// TIA Portal V19 export
DATA_BLOCK "MANUAL"   // DB12
{ S7_Optimized_Access := 'TRUE' }
// stored: MemoryReserve 100
   VAR
      "MGF FEED PUMP WORKING" : Bool;
      "MFG FEED PUMP STANDBY" : Bool;
      "RO FEED PUMP WORKING" : Bool;
      "RO FEED PUMP STANDBY" : Bool;
      "RO HPP PUMP WORKING" : Bool;
      "RO HPP PUMP STANDBY" : Bool;
      "SMBS AGT-1" : Bool;
      "SALT TANK AGT-2" : Bool;
      "RO SMBS AGT-3" : Bool;
      "DP-1" : Bool;
      "DP-2" : Bool;
      "DP-3" : Bool;
      "DP-4" : Bool;
      "DP-5" : Bool;
      "DP-6" : Bool;
      "UV-1-DO" : Bool;
      "UV-2-DO" : Bool;
      HOOTER : Bool;
      "PSFV-1 – OPEN" : Bool;
      "PSFV-1 – CLOSE" : Bool;
      "PSFV-2 – OPEN" : Bool;
      "PSFV-2 – CLOSE" : Bool;
      "PSFV-3 – OPEN" : Bool;
      "PSFV-3 – CLOSE" : Bool;
      "PSFV-4 – OPEN" : Bool;
      "PSFV-4 – CLOSE" : Bool;
      "PSFV-5 – OPEN" : Bool;
      "PSFV-5 – CLOSE" : Bool;
      "PSFV-6 – OPEN" : Bool;
      "PSFV-6 – CLOSE" : Bool;
      "ACFV-1 – OPEN" : Bool;
      "ACFV-1 – CLOSE" : Bool;
      "ACFV-2 – OPEN" : Bool;
      "ACFV-2 – CLOSE" : Bool;
      "ACFV-3 – OPEN" : Bool;
      "ACFV-3 – CLOSE" : Bool;
      "ACFV-4 – OPEN" : Bool;
      "ACFV-4 - CLOSE" : Bool;
      "ACFV-5 – OPEN" : Bool;
      "ACFV-5 – CLOSE" : Bool;
      "ACFV-6 – OPEN" : Bool;
      "ACFV-6 – CLOSE" : Bool;
      "SFV-1 – OPEN" : Bool;
      "SFV-1 – CLOSE" : Bool;
      "SFV-2 – OPEN" : Bool;
      "SFV-2 – CLOSE" : Bool;
      "SFV-3 – OPEN" : Bool;
      "SFV-3 – CLOSE" : Bool;
      "SFV-4 – OPEN" : Bool;
      "SFV-4 – CLOSE" : Bool;
      "SFV-5 – OPEN" : Bool;
      "SFV-5 – CLOSE" : Bool;
      "SFV-6 – OPEN" : Bool;
      "SFV-6 – CLOSE" : Bool;
      "SFV-7 – OPEN" : Bool;
      "SFV-7 – CLOSE" : Bool;
      "SFV-8 – OPEN" : Bool;
      "SFV-8 – CLOSE" : Bool;
      "AV-1 – OPEN" : Bool;
      "AV-1 – CLOSE" : Bool;
      "AV-2 – OPEN" : Bool;
      "AV-2 – CLOSE" : Bool;
      "AV-3 – OPEN" : Bool;
      "AV-3 – CLOSE" : Bool;
      "AV-4 – OPEN" : Bool;
      "AV-4 – CLOSE" : Bool;
      "MANUAL CIP PUMP" : Bool;
      new : Struct
         "RO2 HPP" : Bool;
         "NEW OUTPUTS_PW TRANSFER PUMP S OP" : Bool;
         "NEW OUTPUTS_PW TRANSFER PUMP W OP" : Bool;
      END_STRUCT;
   END_VAR
BEGIN
END_DATA_BLOCK
